INTERFACE I_ContinuousDrive EXTENDS I_Drive

METHOD ABSTRACT moveContinuous : BOOL
VAR_INPUT
	newDirection : MC_Direction;
END_VAR
END_METHOD

END_INTERFACE

(* stored: Version 1.1.0.1, ProductVersion 3.1.4024.11
   Itf I_ContinuousDrive: Id {4acf1163-0cbe-46a9-aeb5-90a0386ec34b}
   Method moveContinuous: Id {35e50634-4dba-44f0-827b-1ffa86f3aaca} *)
